// TIA Portal V15.1 export
// export: Created 2020-06-12T07:35:46.4287109Z, ExportSetting None, DisplayName Totally Integrated Automation Portal, DisplayVersion V15.1, DisplayName TIA Portal Openness, DisplayVersion V15.1, DisplayName STEP 7 Professional, DisplayVersion V15.1, DisplayName STEP 7 Safety, DisplayVersion V15.1, DisplayName WinCC Advanced, DisplayVersion V15.1
FUNCTION_BLOCK "Single_Vessel"   // FB13, SCL
{ S7_Optimized_Access := 'TRUE' }
// stored: MemoryReserve 100, SetENOAutomatically False
   VAR_INPUT
      iStartCycle { ExternalAccessible := 'False'; ExternalVisible := 'False'; ExternalWritable := 'False'} : Bool;   // Start Alloy Sequence
      iReset_Error { ExternalAccessible := 'False'; ExternalVisible := 'False'; ExternalWritable := 'False'} : Bool;
      iMotorReady { ExternalAccessible := 'False'; ExternalVisible := 'False'; ExternalWritable := 'False'} : Bool;   // Vibro-Motor Ready
      IMotorRunning { ExternalAccessible := 'False'; ExternalVisible := 'False'; ExternalWritable := 'False'} : Bool;
      iSkip1 { ExternalAccessible := 'False'; ExternalVisible := 'False'; ExternalWritable := 'False'} : Bool;
      iSkip2 { ExternalAccessible := 'False'; ExternalVisible := 'False'; ExternalWritable := 'False'} : Bool;
      iWeight_per_Cycle { ExternalAccessible := 'False'; ExternalVisible := 'False'; ExternalWritable := 'False'} : Real;   // Setvalue of vessel in g/min
      iSlowSpeed_Setvalue { ExternalAccessible := 'False'; ExternalVisible := 'False'; ExternalWritable := 'False'} : Real;   // Setvalue for slow speed
      iFastSpeed_Setvalue { ExternalAccessible := 'False'; ExternalVisible := 'False'; ExternalWritable := 'False'} : Real;   // Setvalue for high speed
      iScaleValue { ExternalAccessible := 'False'; ExternalVisible := 'False'; ExternalWritable := 'False'} : Real;   // Aktuelles Gewicht in der Wägeschale in g
   END_VAR
   VAR_OUTPUT
      oActivateMotor { ExternalAccessible := 'False'; ExternalVisible := 'False'; ExternalWritable := 'False'} : Bool;   // Output to Motor
      oMotorSetValue { ExternalAccessible := 'False'; ExternalVisible := 'False'; ExternalWritable := 'False'} : Real;   // Speed set value for motor
      oCycleFinished { ExternalAccessible := 'False'; ExternalVisible := 'False'; ExternalWritable := 'False'} : Bool;   // Finished the sequence
      oError { ExternalAccessible := 'False'; ExternalVisible := 'False'; ExternalWritable := 'False'} : Bool;   // Error, max time needed
   END_VAR
   VAR_IN_OUT
      HMI_data : "Alloy_Vesel_HMI";   // Data to HMI
   END_VAR
   VAR
      StateID { ExternalAccessible := 'False'; ExternalVisible := 'False'; ExternalWritable := 'False'} : Int;   // Seuence ID
      WeighingActive { ExternalAccessible := 'False'; ExternalVisible := 'False'; ExternalWritable := 'False'} : Bool;   // sequence is active
      WeightStart { ExternalAccessible := 'False'; ExternalVisible := 'False'; ExternalWritable := 'False'} : Real;   // Start weight at beginning
      WeightEnd { ExternalAccessible := 'False'; ExternalVisible := 'False'; ExternalWritable := 'False'} : Real;   // Calculated weight where motor should stop
      WeightDifference { ExternalAccessible := 'False'; ExternalVisible := 'False'; ExternalWritable := 'False'} : Real;   // Difference between calculated and measured weight
      WeightEnd_Measured { ExternalAccessible := 'False'; ExternalVisible := 'False'; ExternalWritable := 'False'} : Real;   // Weight measured at end of motor feeding
      _StartCycle { ExternalAccessible := 'False'; ExternalVisible := 'False'; ExternalWritable := 'False'} : Bool;   // Temp to recognize flank
      Timer_Wait_Scale { ExternalAccessible := 'False'; ExternalVisible := 'False'; ExternalWritable := 'False'} : TON_TIME;   // Timer wait to stabilize scale
      Timer_Cycle_Error { ExternalAccessible := 'False'; ExternalVisible := 'False'; ExternalWritable := 'False'} : TON_TIME;   // Timer max time for sequence
   END_VAR
   VAR_TEMP
      tSkipStart : Bool;   // Skip start of vessel
   END_VAR
BEGIN
   // Reset Error
   IF #iReset_Error = true THEN
       #oActivateMotor := false;
       #HMI_data.Weight_Sum_AllCycles := 0;
       #StateID := 0;
       #_StartCycle := false;
       #oError := false;
       #HMI_data.Status_Error := false;
       #HMI_data.Cycle_Count := 0;
       #HMI_data.Weight_Difference := 0;
       #Timer_Cycle_Error(IN := false,
                          PT := t#0s);
   END_IF;

   /////////////////////////////////////////////////////////////////////////////////////////////////// 
   //Check the cycle length and generate alarm if it takes too much time
   /////////////////////////////////////////////////////////////////////////////////////////////////// 
   #Timer_Cycle_Error(IN := #WeighingActive,
                      PT := #HMI_data.TimeCycleError);

   IF #Timer_Cycle_Error.Q = true THEN
       #WeighingActive := false;
       #oActivateMotor := false;
       #StateID := -2;
       #oError := #Timer_Cycle_Error.Q;
       #HMI_data.Status_Error := true;
       RETURN;
   END_IF;

   /////////////////////////////////////////////////////////////////////////////////////////////////// 
   //Wait for rising edge on iStart_Cycle
   /////////////////////////////////////////////////////////////////////////////////////////////////// 
   IF #iStartCycle = false THEN
       #_StartCycle := false;
       #oCycleFinished := false;
       #oError := false;
       #HMI_data.Status_Error := false;
   END_IF;
   IF #iStartCycle = true AND #_StartCycle = false THEN
       #_StartCycle := true;
       #WeighingActive := true;
       #oCycleFinished := false;
       #StateID := 0;
   END_IF;

   /////////////////////////////////////////////////////////////////////////////////////////////////// 
   //Begin step sequence
   /////////////////////////////////////////////////////////////////////////////////////////////////// 
   //Standby, check start conditions
   /////////////////////////////////////////////////////////////////////////////////////////////////// 
   IF #StateID = 0 THEN
       #tSkipStart := false;

       IF #HMI_data.Weight_Set_perCycle = 0 THEN
           #tSkipStart := true;
       END_IF;

       // "MELT_VAR_DB".meas_ingot_WT > 0 AND  "MELT_VAR_DB".meas_ingot_WT < #HMI_data.StartAlloy
       IF #iSkip1 THEN
           #tSkipStart := true;
       END_IF;

       // "MELT_VAR_DB".meas_ingot_WT > 0 AND "MELT_VAR_DB".meas_ingot_WT > #HMI_data.StopAlloy
       IF #iSkip2 THEN
           #tSkipStart := true;
       END_IF;

       IF #tSkipStart = true THEN
           #WeighingActive := false;
           #oCycleFinished := true;
           #_StartCycle := false;
           #oActivateMotor := false;
           #StateID := 0;
           RETURN;
       END_IF;

       #oActivateMotor := false;
       #oMotorSetValue := 0;

       #StateID := 1;
       RETURN;
   END_IF;


   /////////////////////////////////////////////////////////////////////////////////////////////////// 
   //Calculate values for start
   /////////////////////////////////////////////////////////////////////////////////////////////////// 
   IF #StateID = 1 THEN
       //If Vessel is deactivated go to end (Vessel SetWeight = 0)
       IF #iWeight_per_Cycle = 0 THEN
           #WeightEnd := 0;
           #WeightStart := 0;
           #StateID := 10;
           RETURN;
       END_IF;

       #WeightStart := #iScaleValue;
       #WeightEnd := #WeightStart + #iWeight_per_Cycle + #WeightDifference;


       //If last cycle feeded to much alloy addition, skip this cycle
       IF #WeightEnd < #WeightStart THEN
           #WeightDifference := #WeightDifference + #iWeight_per_Cycle;
           #HMI_data.Weight_Difference := #WeightDifference;
           #HMI_data.Cycle_Count := #HMI_data.Cycle_Count + 1;

           #WeighingActive := false;
           #oCycleFinished := true;
           #_StartCycle := false;
           #StateID := 0;
           RETURN;
       END_IF;

       #StateID := 2;
       RETURN;
   END_IF;

   /////////////////////////////////////////////////////////////////////////////////////////////////// 
   //Activate Motor and begin weighing
   /////////////////////////////////////////////////////////////////////////////////////////////////// 
   IF #StateID = 2 THEN
       IF #iMotorReady = true THEN
           #oMotorSetValue := #iFastSpeed_Setvalue;
           #oActivateMotor := true;
           #StateID := 3;
           RETURN;
       END_IF;
   END_IF;

   /////////////////////////////////////////////////////////////////////////////////////////////////// 
   //Wait until calculated weight is reached
   /////////////////////////////////////////////////////////////////////////////////////////////////// 
   IF #StateID = 3 THEN
       // Set speed for Vibro Motor
       IF #iScaleValue > #WeightEnd - #HMI_data.WeightSpeedReduction THEN
           #oMotorSetValue := #iSlowSpeed_Setvalue;
       ELSE
           #oMotorSetValue := #iFastSpeed_Setvalue;
       END_IF;

       //Motor Ready Error
       // IF #iMotorReady = false THEN
       //     #StateID := -2;
       // END_IF;


       //Shut off Motor when calculated weight on scale is reached
       IF #iScaleValue > #WeightEnd - #HMI_data.WeightPreStop  THEN
           #oActivateMotor := false;

           #HMI_data.Weight_Difference := #WeightDifference;

           //Reset Timer for stable scale measurement
           #Timer_Wait_Scale(IN := false,
                             PT := t#0s);

           #StateID := 4;
           RETURN;
       END_IF;
   END_IF;

   /////////////////////////////////////////////////////////////////////////////////////////////////// 
   //Wait for stabilize timer until scale measurement is stable
   /////////////////////////////////////////////////////////////////////////////////////////////////// 
   IF #StateID = 4 THEN
       #Timer_Wait_Scale(IN := true,
                         PT := #HMI_data.TimeMeasurementStabilize);

       IF #Timer_Wait_Scale.Q = true THEN
           #WeightEnd_Measured := #iScaleValue;

           #StateID := 5;
           RETURN;
       END_IF;
   END_IF;


   /////////////////////////////////////////////////////////////////////////////////////////////////// 
   //Calculate the difference between real weight and calculated weight
   /////////////////////////////////////////////////////////////////////////////////////////////////// 
   IF #StateID = 5 THEN
       #WeightDifference := #WeightEnd - #WeightEnd_Measured;
       #StateID := 10;
       RETURN;
   END_IF;


   /////////////////////////////////////////////////////////////////////////////////////////////////// 
   //End of cycle
   /////////////////////////////////////////////////////////////////////////////////////////////////// 
   IF #StateID = 10 THEN
       #HMI_data.Weight_Sum_AllCycles := #HMI_data.Weight_Sum_AllCycles + (#WeightEnd_Measured - #WeightStart);

       #HMI_data.Cycle_Count := #HMI_data.Cycle_Count + 1;

       #WeighingActive := false;
       #oCycleFinished := true;
       #_StartCycle := false;

       #HMI_data.Weight_Difference := #WeightDifference;

       #StateID := 0;
       RETURN;
   END_IF;
END_FUNCTION_BLOCK
